// TIA Portal V20 export
// export: Created 2025-12-01T14:57:36.0041783Z, ExportSetting None, DisplayName Totally Integrated Automation Portal, DisplayVersion V20 Update 3, DisplayName TIA Portal Openness, DisplayVersion V20 Update 3, DisplayName TIA Portal Version Control Interface, DisplayVersion V20 Update 3, DisplayName STEP 7 Professional, DisplayVersion V20 Update 3, DisplayName STEP 7 Safety, DisplayVersion V20 Update 2, DisplayName WinCC Basic/Comfort/Advanced, DisplayVersion V20 Update 3, DisplayName WinCC Professional, DisplayVersion V20 Update 3, DisplayName WinCC Unified, DisplayVersion V20 Update 3
FUNCTION_BLOCK "FB984_Control_i950_ELEV / VTD"   // FB984, LAD
{ S7_Optimized_Access := 'FALSE' }
// stored: AutoNumber false, SetENOAutomatically false
   VAR_INPUT
      NumDispositivo : UInt;   // Numero de Maquina
      Error_Tx : Bool;
      Protusion : Bool;
      OrdenPosicion : Bool;
      "Avance-Subir" : Bool;
      "Retroceso-Bajar" : Bool;
      ConsignaPosicion : Real;
      SHome_Available : Bool;
      SHome_Activated : Bool;
   END_VAR
   VAR_OUTPUT
      PosicionActual : Real;
      VelocidadActual : Real;   // Velocidad Actual
      EnPosicion : Bool;   // Posicion OK de la Orden
      SHome_Start : Bool;   // Inicio Homing de la tarjeta SRM
      SHome_Load : Bool;   // Confirmacion de la tarjeta SRM
      Freno : Bool;
   END_VAR
   VAR
      TMP_Rearme { S7_SetPoint := 'True'} : TOF_TIME;
      TEspera_ET04Ref { S7_SetPoint := 'True'} : TON_TIME;
      TEspera_ET05Ref { S7_SetPoint := 'True'} : TON_TIME;
      TEspera_ET00 { S7_SetPoint := 'True'} : TON_TIME;
      PosicionOrden { S7_SetPoint := 'True'} : Real;
      ConsignaVelocidad : Real;
      ET_00 { S7_SetPoint := 'True'} : Bool;
      ET_01 : Bool;
      ET_02 : Bool;
      ET_03Ref : Bool;
      ET_04Ref : Bool;
      ET_05Ref : Bool;
      ET_06Ref : Bool;
      Rem_MesaDestino : UInt;
   END_VAR
   VAR_TEMP
      EstadoZona : "EstadoZona";   // Estado de la Zona
      EstadoMAQ : "EstadoMaquina_Variador_i950";
      NumMaquina : UInt;
      Byte0 : Int;
      Byte1 : Int;
      Byte2 : Int;
      Byte3 : Int;
      Direccion_Pos_Actual : DInt;
      Direccion_Velocity : DInt;
      Direccion_Position : DInt;
      DireccionCorriente : DInt;
      Acele : DInt;
      Dece : DInt;
      Jerk : DInt;
      Torque : DInt;
      DirInicial : Int;   // Dirección inicio periferia
      "ACC (m/s2)" : Real;
      "DCC(m/s2)" : Real;
      "VelocidadAuto(m/s)" : Real;
      "VelocidadHoming(m/s)" : Real;
      "PosicionHorming(mm)" : Real;
      VarReal : Real;
      Nodo : Int;   // Numero de Maquina
      VReal : DWord;
      VelocityAuto : DInt;
      VelocityHoming : DInt;
   END_VAR
   VAR_TEMP   // added for the SCL form of the ladder/FBD networks
      _w1 : Bool;
   END_VAR
BEGIN

REGION Network 1: Recoger Variables
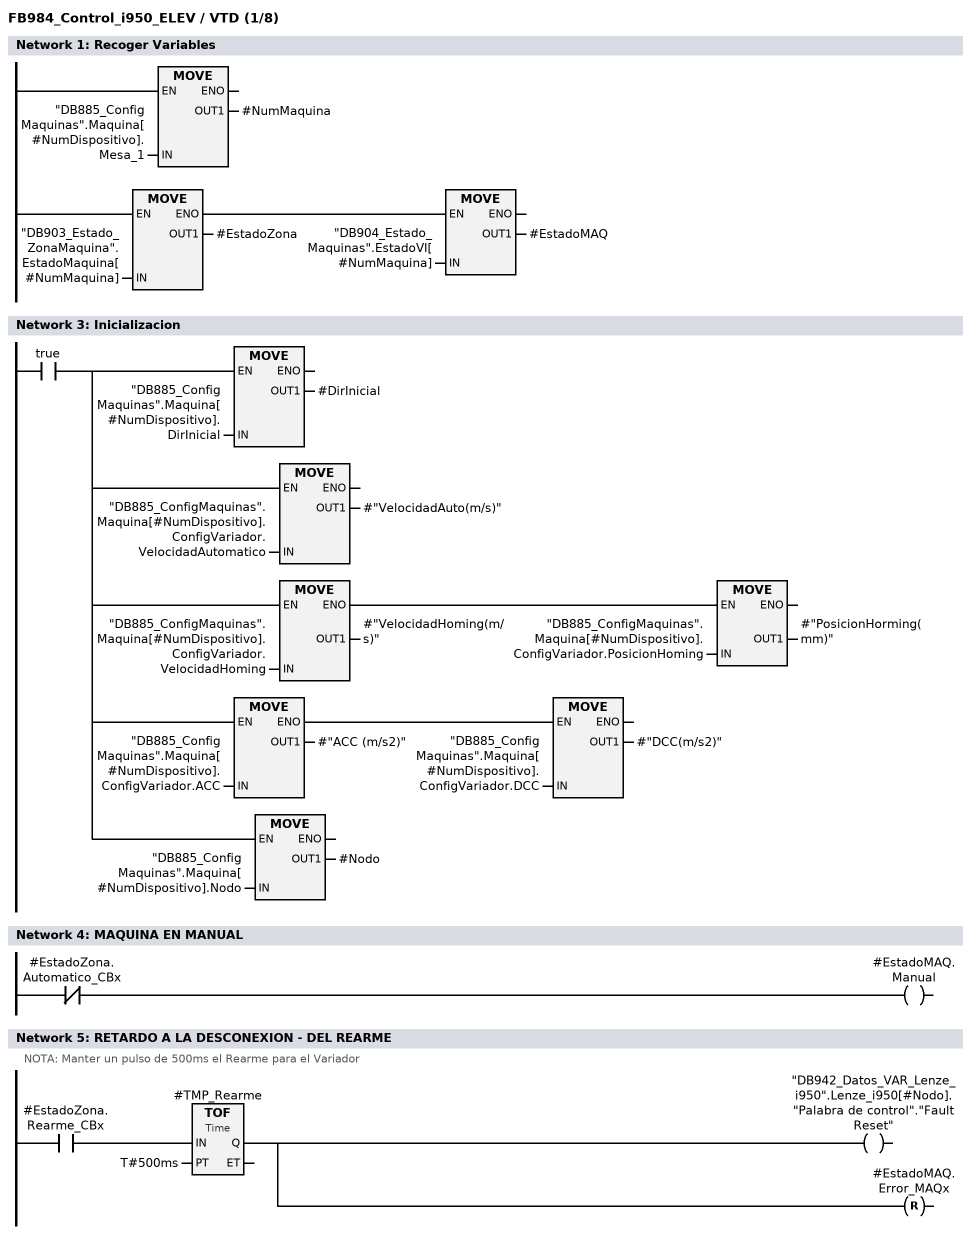
   RUNG wire#powerrail
      Move(in := "DB885_ConfigMaquinas".Maquina[#NumDispositivo].Mesa_1, out1 => #NumMaquina)
   END_RUNG
   RUNG wire#powerrail
      Move(in := "DB903_Estado_ZonaMaquina".EstadoMaquina[#NumMaquina], out1 => #EstadoZona)
      Move(in := "DB904_Estado_Maquinas".EstadoVI[#NumMaquina], out1 => #EstadoMAQ)
   END_RUNG
   // the same network as SCL:
   #NumMaquina := "DB885_ConfigMaquinas".Maquina[#NumDispositivo].Mesa_1;
   #EstadoZona := "DB903_Estado_ZonaMaquina".EstadoMaquina[#NumMaquina];
   #EstadoMAQ := "DB904_Estado_Maquinas".EstadoVI[#NumMaquina];
END_REGION

REGION Network 2: >>>>>>>>>>>>>>>>>>>>>>>>>>>>>>>>>>>>>>>>>>>>>>>>>>>>>>>>>>>>>>>>>>>>>>>
END_REGION

REGION Network 3: Inicializacion
   RUNG wire#powerrail
      Contact( true )
      wire#w1
      Move(in := "DB885_ConfigMaquinas".Maquina[#NumDispositivo].DirInicial, out1 => #DirInicial)
   END_RUNG
   RUNG wire#w1
      Move(in := "DB885_ConfigMaquinas".Maquina[#NumDispositivo].ConfigVariador.VelocidadAutomatico, out1 => #"VelocidadAuto(m/s)")
   END_RUNG
   RUNG wire#w1
      Move(in := "DB885_ConfigMaquinas".Maquina[#NumDispositivo].ConfigVariador.VelocidadHoming, out1 => #"VelocidadHoming(m/s)")
      Move(in := "DB885_ConfigMaquinas".Maquina[#NumDispositivo].ConfigVariador.PosicionHoming, out1 => #"PosicionHorming(mm)")
   END_RUNG
   RUNG wire#w1
      Move(in := "DB885_ConfigMaquinas".Maquina[#NumDispositivo].ConfigVariador.ACC, out1 => #"ACC (m/s2)")
      Move(in := "DB885_ConfigMaquinas".Maquina[#NumDispositivo].ConfigVariador.DCC, out1 => #"DCC(m/s2)")
   END_RUNG
   RUNG wire#w1
      Move(in := "DB885_ConfigMaquinas".Maquina[#NumDispositivo].Nodo, out1 => #Nodo)
   END_RUNG
   // the same network as SCL:
   IF true THEN
       #DirInicial := "DB885_ConfigMaquinas".Maquina[#NumDispositivo].DirInicial;
       #"VelocidadAuto(m/s)" := "DB885_ConfigMaquinas".Maquina[#NumDispositivo].ConfigVariador.VelocidadAutomatico;
       #"VelocidadHoming(m/s)" := "DB885_ConfigMaquinas".Maquina[#NumDispositivo].ConfigVariador.VelocidadHoming;
       #"PosicionHorming(mm)" := "DB885_ConfigMaquinas".Maquina[#NumDispositivo].ConfigVariador.PosicionHoming;
       #"ACC (m/s2)" := "DB885_ConfigMaquinas".Maquina[#NumDispositivo].ConfigVariador.ACC;
       #"DCC(m/s2)" := "DB885_ConfigMaquinas".Maquina[#NumDispositivo].ConfigVariador.DCC;
       #Nodo := "DB885_ConfigMaquinas".Maquina[#NumDispositivo].Nodo;
   END_IF;
END_REGION

REGION Network 4: MAQUINA EN MANUAL
   RUNG wire#powerrail
      I_Contact( #EstadoZona.Automatico_CBx )
      Coil( #EstadoMAQ.Manual )
   END_RUNG
   // the same network as SCL:
   #EstadoMAQ.Manual := NOT #EstadoZona.Automatico_CBx;
END_REGION

REGION Network 5: RETARDO A LA DESCONEXION - DEL REARME
   // NOTA: Manter un pulso de 500ms el Rearme para el Variador
   RUNG wire#powerrail
      Contact( #EstadoZona.Rearme_CBx )
      { S7_Templates := "time_type := Time" } #TMP_Rearme.TOF(pt := T#500ms, et =>)
      wire#w1
      Coil( "DB942_Datos_VAR_Lenze_i950".Lenze_i950[#Nodo]."Palabra de control"."Fault Reset" )
   END_RUNG
   RUNG wire#w1
      R_Coil( #EstadoMAQ.Error_MAQx )
   END_RUNG
   // the same network as SCL:
   #TMP_Rearme(IN := #EstadoZona.Rearme_CBx, PT := T#500ms);   // TOF
   "DB942_Datos_VAR_Lenze_i950".Lenze_i950[#Nodo]."Palabra de control"."Fault Reset" := #TMP_Rearme.Q;
   IF #TMP_Rearme.Q THEN #EstadoMAQ.Error_MAQx := FALSE; END_IF;
END_REGION

REGION Network 6 (SCL): Direcciones
   #Byte0 := #DirInicial;
   #Byte1 := #DirInicial + 1;
   #Byte2 := #DirInicial + 2;
   #Byte3 := #DirInicial + 3;
   #Direccion_Pos_Actual := #DirInicial + 12;
   #Direccion_Velocity := #DirInicial + 8;
   #Direccion_Position := #DirInicial + 12;
   #DireccionCorriente := #DirInicial + 24;
   #Acele := #DirInicial + 16;
   #Dece := #DirInicial + 20;
   #Jerk := #DirInicial + 24;
   #Torque := #DirInicial + 28;
END_REGION

REGION Network 7 (SCL): Lectura de variables del Variador
   //Leo las variables que nos interesan

   "DB942_Datos_VAR_Lenze_i950".Lenze_i950[#Nodo]."Estatus variador"."Positioning Profile Done" := PEEK_BOOL(area := 16#81, dbNumber := 0, byteOffset := #Byte1, bitOffset := 5);
   "DB942_Datos_VAR_Lenze_i950".Lenze_i950[#Nodo]."Estatus variador"."Target Reached" := PEEK_BOOL(area := 16#81, dbNumber := 0, byteOffset := #Byte2, bitOffset := 2);
   "DB942_Datos_VAR_Lenze_i950".Lenze_i950[#Nodo]."Estatus variador"."STO Active" := PEEK_BOOL(area := 16#81, dbNumber := 0, byteOffset := #Byte2, bitOffset := 7);
   "DB942_Datos_VAR_Lenze_i950".Lenze_i950[#Nodo]."Estatus variador"."Operation Enabled" := PEEK_BOOL(area := 16#81, dbNumber := 0, byteOffset := #Byte3, bitOffset := 2);
   "DB942_Datos_VAR_Lenze_i950".Lenze_i950[#Nodo]."Estatus variador"."Drive Fault" := PEEK_BOOL(area := 16#81, dbNumber := 0, byteOffset := #Byte3, bitOffset := 3);
   "DB942_Datos_VAR_Lenze_i950".Lenze_i950[#Nodo]."Estatus variador"."Drive Homed" := PEEK_BOOL(area := 16#81, dbNumber := 0, byteOffset := #Byte3, bitOffset := 4);
   "DB942_Datos_VAR_Lenze_i950".Lenze_i950[#Nodo]."Estatus variador"."Jogging Busy" := PEEK_BOOL(area := 16#81, dbNumber := 0, byteOffset := #Byte3, bitOffset := 6);
   "DB942_Datos_VAR_Lenze_i950".Lenze_i950[#Nodo].Velocity := PEEK_DWORD(area := 16#81, dbNumber := 0, byteOffset := #Direccion_Velocity);
   "DB942_Datos_VAR_Lenze_i950".Lenze_i950[#Nodo].Actual_Position := PEEK_DWORD(area := 16#81, dbNumber := 0, byteOffset := #Direccion_Pos_Actual);
   "DB942_Datos_VAR_Lenze_i950".Lenze_i950[#Nodo]."Corriente%" := PEEK_DWORD(area := 16#81, dbNumber := 0, byteOffset := #DireccionCorriente);
END_REGION

REGION Network 8: Captura de la corriente
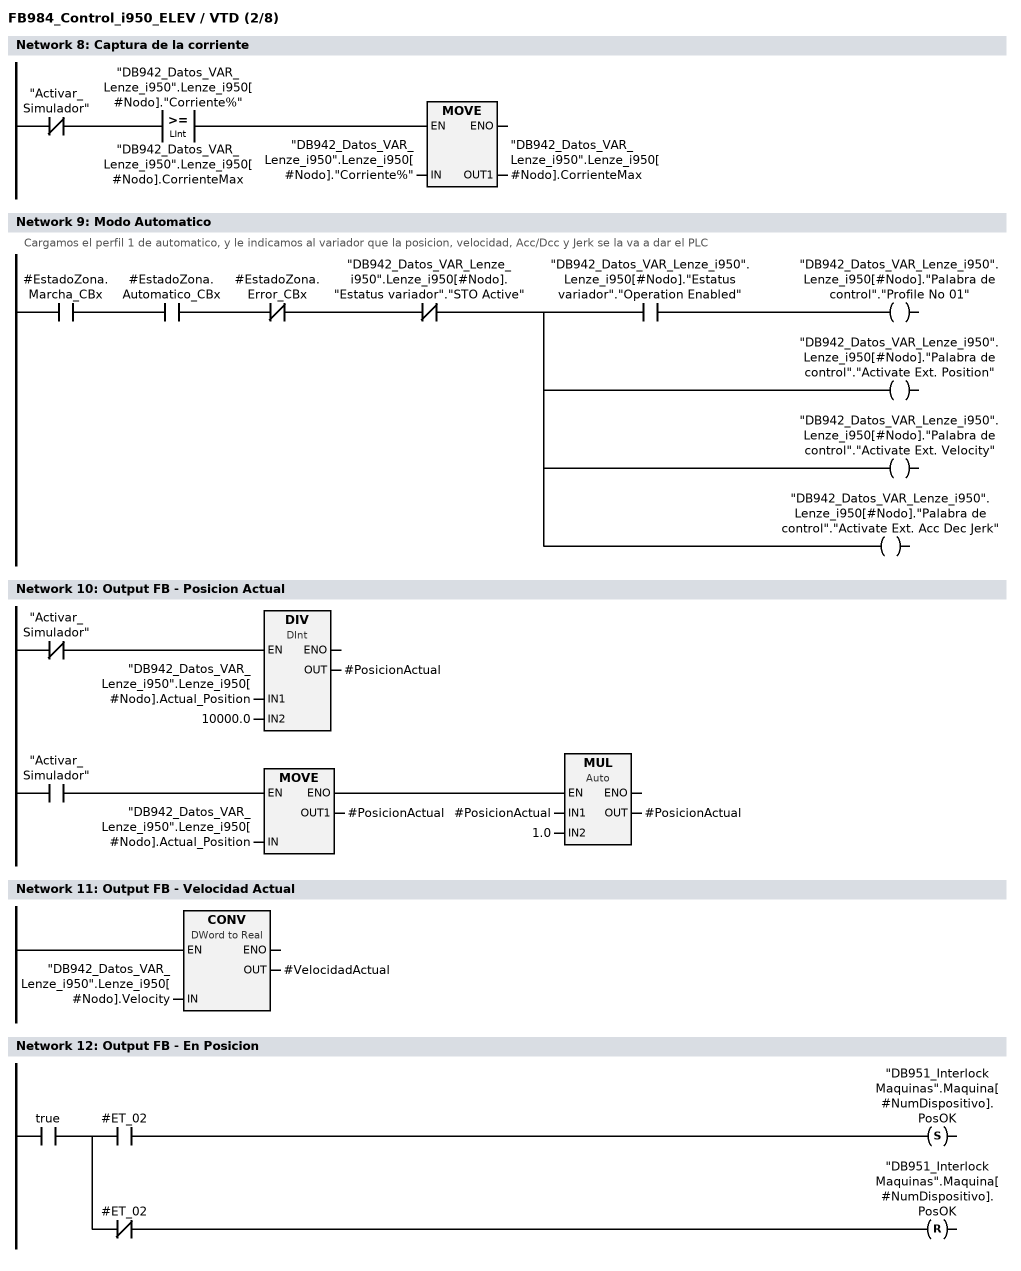
   RUNG wire#powerrail
      I_Contact( "Activar_Simulador" )
      { S7_Templates := "SrcType := LInt" } GE_Contact(in1 := "DB942_Datos_VAR_Lenze_i950".Lenze_i950[#Nodo]."Corriente%", in2 := "DB942_Datos_VAR_Lenze_i950".Lenze_i950[#Nodo].CorrienteMax)
      Move(in := "DB942_Datos_VAR_Lenze_i950".Lenze_i950[#Nodo]."Corriente%", out1 => "DB942_Datos_VAR_Lenze_i950".Lenze_i950[#Nodo].CorrienteMax)
   END_RUNG
   // the same network as SCL:
   IF NOT "Activar_Simulador" AND ("DB942_Datos_VAR_Lenze_i950".Lenze_i950[#Nodo]."Corriente%" >= "DB942_Datos_VAR_Lenze_i950".Lenze_i950[#Nodo].CorrienteMax) THEN
       "DB942_Datos_VAR_Lenze_i950".Lenze_i950[#Nodo].CorrienteMax := "DB942_Datos_VAR_Lenze_i950".Lenze_i950[#Nodo]."Corriente%";
   END_IF;
END_REGION

REGION Network 9: Modo Automatico
   // Cargamos el perfil 1 de automatico, y le indicamos al variador que la posicion, velocidad, Acc/Dcc y Jerk se la va a dar el PLC
   RUNG wire#powerrail
      Contact( #EstadoZona.Marcha_CBx )
      Contact( #EstadoZona.Automatico_CBx )
      I_Contact( #EstadoZona.Error_CBx )
      I_Contact( "DB942_Datos_VAR_Lenze_i950".Lenze_i950[#Nodo]."Estatus variador"."STO Active" )
      wire#w1
      Contact( "DB942_Datos_VAR_Lenze_i950".Lenze_i950[#Nodo]."Estatus variador"."Operation Enabled" )
      Coil( "DB942_Datos_VAR_Lenze_i950".Lenze_i950[#Nodo]."Palabra de control"."Profile No 01" )
   END_RUNG
   RUNG wire#w1
      Coil( "DB942_Datos_VAR_Lenze_i950".Lenze_i950[#Nodo]."Palabra de control"."Activate Ext. Position" )
   END_RUNG
   RUNG wire#w1
      Coil( "DB942_Datos_VAR_Lenze_i950".Lenze_i950[#Nodo]."Palabra de control"."Activate Ext. Velocity" )
   END_RUNG
   RUNG wire#w1
      Coil( "DB942_Datos_VAR_Lenze_i950".Lenze_i950[#Nodo]."Palabra de control"."Activate Ext. Acc Dec Jerk" )
   END_RUNG
   // the same network as SCL:
   #_w1 := #EstadoZona.Marcha_CBx AND #EstadoZona.Automatico_CBx AND NOT #EstadoZona.Error_CBx AND NOT "DB942_Datos_VAR_Lenze_i950".Lenze_i950[#Nodo]."Estatus variador"."STO Active";
   "DB942_Datos_VAR_Lenze_i950".Lenze_i950[#Nodo]."Palabra de control"."Profile No 01" := #_w1 AND "DB942_Datos_VAR_Lenze_i950".Lenze_i950[#Nodo]."Estatus variador"."Operation Enabled";
   "DB942_Datos_VAR_Lenze_i950".Lenze_i950[#Nodo]."Palabra de control"."Activate Ext. Position" := #_w1;
   "DB942_Datos_VAR_Lenze_i950".Lenze_i950[#Nodo]."Palabra de control"."Activate Ext. Velocity" := #_w1;
   "DB942_Datos_VAR_Lenze_i950".Lenze_i950[#Nodo]."Palabra de control"."Activate Ext. Acc Dec Jerk" := #_w1;
END_REGION

REGION Network 10: Output FB - Posicion Actual
   RUNG wire#powerrail
      I_Contact( "Activar_Simulador" )
      { S7_Templates := "SrcType := DInt" } Div(in1 := "DB942_Datos_VAR_Lenze_i950".Lenze_i950[#Nodo].Actual_Position, in2 := 10000.0, out => #PosicionActual)
   END_RUNG
   RUNG wire#powerrail
      Contact( "Activar_Simulador" )
      Move(in := "DB942_Datos_VAR_Lenze_i950".Lenze_i950[#Nodo].Actual_Position, out1 => #PosicionActual)
      Mul(in1 := #PosicionActual, in2 := 1.0, out => #PosicionActual)
   END_RUNG
   // the same network as SCL:
   IF NOT "Activar_Simulador" THEN
       #PosicionActual := "DB942_Datos_VAR_Lenze_i950".Lenze_i950[#Nodo].Actual_Position / 10000.0;
   END_IF;
   IF "Activar_Simulador" THEN
       #PosicionActual := "DB942_Datos_VAR_Lenze_i950".Lenze_i950[#Nodo].Actual_Position;
       #PosicionActual := #PosicionActual * 1.0;
   END_IF;
END_REGION

REGION Network 11: Output FB - Velocidad Actual
   RUNG wire#powerrail
      { S7_Templates := "[SrcType := DWord, DestType := Real]" } Convert(in := "DB942_Datos_VAR_Lenze_i950".Lenze_i950[#Nodo].Velocity, out => #VelocidadActual)
   END_RUNG
   // the same network as SCL:
   #VelocidadActual := DWORD_TO_REAL("DB942_Datos_VAR_Lenze_i950".Lenze_i950[#Nodo].Velocity);
END_REGION

REGION Network 12: Output FB - En Posicion
   RUNG wire#powerrail
      Contact( true )
      wire#w1
      Contact( #ET_02 )
      S_Coil( "DB951_InterlockMaquinas".Maquina[#NumDispositivo].PosOK )
   END_RUNG
   RUNG wire#w1
      I_Contact( #ET_02 )
      R_Coil( "DB951_InterlockMaquinas".Maquina[#NumDispositivo].PosOK )
   END_RUNG
   // the same network as SCL:
   IF true AND #ET_02 THEN "DB951_InterlockMaquinas".Maquina[#NumDispositivo].PosOK := TRUE; END_IF;
   IF true AND NOT #ET_02 THEN "DB951_InterlockMaquinas".Maquina[#NumDispositivo].PosOK := FALSE; END_IF;
END_REGION

REGION Network 13: Consigna de Velocidad
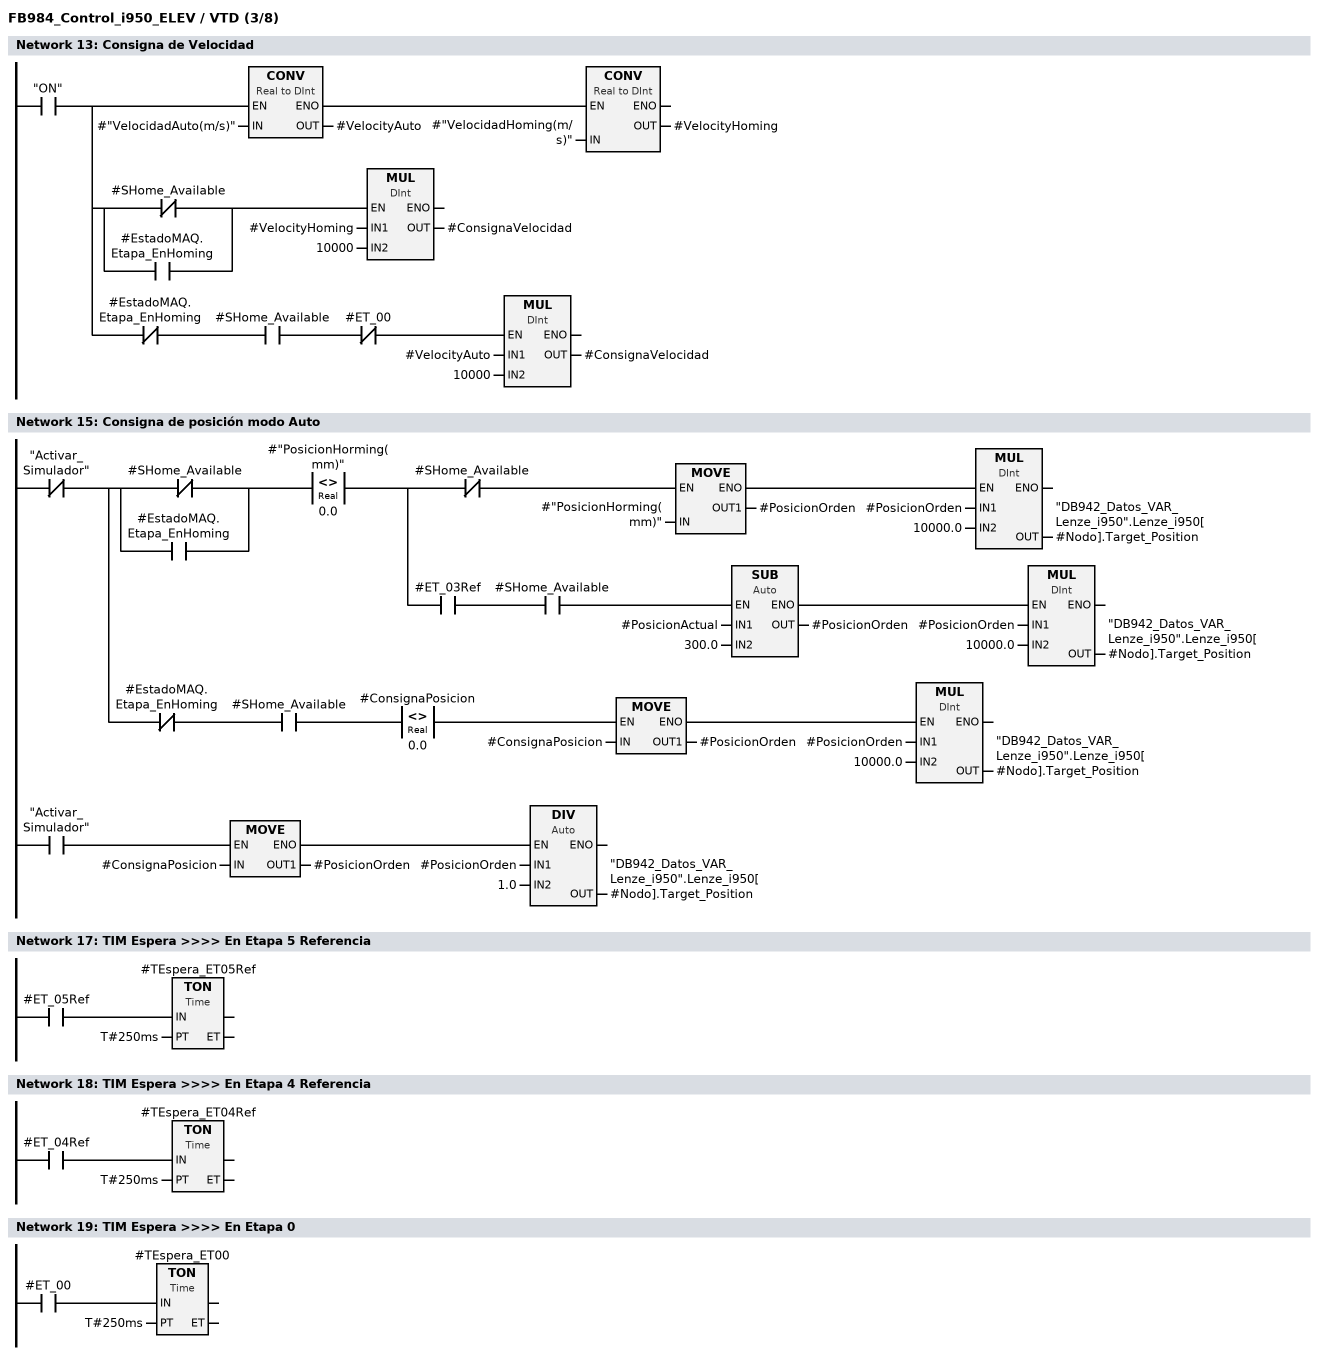
   RUNG wire#powerrail
      Contact( "ON" )
      wire#w1
      { S7_Templates := "[SrcType := Real, DestType := DInt]" } Convert(in := #"VelocidadAuto(m/s)", out => #VelocityAuto)
      { S7_Templates := "[SrcType := Real, DestType := DInt]" } Convert(in := #"VelocidadHoming(m/s)", out => #VelocityHoming)
   END_RUNG
   RUNG wire#w1
      I_Contact( #SHome_Available )
      wire#w2
      { S7_Templates := "SrcType := DInt" } Mul(in1 := #VelocityHoming, in2 := 10000, out => #ConsignaVelocidad)
   END_RUNG
   RUNG wire#w1
      Contact( #EstadoMAQ.Etapa_EnHoming )
   END_RUNG wire#w2
   RUNG wire#w1
      I_Contact( #EstadoMAQ.Etapa_EnHoming )
      Contact( #SHome_Available )
      I_Contact( #ET_00 )
      { S7_Templates := "SrcType := DInt" } Mul(in1 := #VelocityAuto, in2 := 10000, out => #ConsignaVelocidad)
   END_RUNG
   // the same network as SCL:
   IF "ON" THEN
       #VelocityAuto := REAL_TO_DINT(#"VelocidadAuto(m/s)");
       #VelocityHoming := REAL_TO_DINT(#"VelocidadHoming(m/s)");
   END_IF;
   IF "ON" AND (NOT #SHome_Available OR #EstadoMAQ.Etapa_EnHoming) THEN
       #ConsignaVelocidad := #VelocityHoming * 10000;
   END_IF;
   IF "ON" AND NOT #EstadoMAQ.Etapa_EnHoming AND #SHome_Available AND NOT #ET_00 THEN
       #ConsignaVelocidad := #VelocityAuto * 10000;
   END_IF;
END_REGION

REGION Network 14 (SCL): Aceleración y Deceleración
   "DB942_Datos_VAR_Lenze_i950".Lenze_i950[#Nodo].ACC := REAL_TO_DINT (#"ACC (m/s2)" * 100);
   "DB942_Datos_VAR_Lenze_i950".Lenze_i950[#Nodo].DCC  := REAL_TO_DINT(#"DCC(m/s2)" * 100);
END_REGION

REGION Network 15: Consigna de posición modo Auto
   RUNG wire#powerrail
      I_Contact( "Activar_Simulador" )
      wire#w1
      I_Contact( #SHome_Available )
      wire#w2
      { S7_Templates := "SrcType := Real" } NE_Contact(in1 := #"PosicionHorming(mm)", in2 := 0.0)
      wire#w3
      I_Contact( #SHome_Available )
      Move(in := #"PosicionHorming(mm)", out1 => #PosicionOrden)
      { S7_Templates := "SrcType := DInt" } Mul(in1 := #PosicionOrden, in2 := 10000.0, out => "DB942_Datos_VAR_Lenze_i950".Lenze_i950[#Nodo].Target_Position)
   END_RUNG
   RUNG wire#w1
      Contact( #EstadoMAQ.Etapa_EnHoming )
   END_RUNG wire#w2
   RUNG wire#w3
      Contact( #ET_03Ref )
      Contact( #SHome_Available )
      Sub(in1 := #PosicionActual, in2 := 300.0, out => #PosicionOrden)
      { S7_Templates := "SrcType := DInt" } Mul(in1 := #PosicionOrden, in2 := 10000.0, out => "DB942_Datos_VAR_Lenze_i950".Lenze_i950[#Nodo].Target_Position)
   END_RUNG
   RUNG wire#w1
      I_Contact( #EstadoMAQ.Etapa_EnHoming )
      Contact( #SHome_Available )
      { S7_Templates := "SrcType := Real" } NE_Contact(in1 := #ConsignaPosicion, in2 := 0.0)
      Move(in := #ConsignaPosicion, out1 => #PosicionOrden)
      { S7_Templates := "SrcType := DInt" } Mul(in1 := #PosicionOrden, in2 := 10000.0, out => "DB942_Datos_VAR_Lenze_i950".Lenze_i950[#Nodo].Target_Position)
   END_RUNG
   RUNG wire#powerrail
      Contact( "Activar_Simulador" )
      Move(in := #ConsignaPosicion, out1 => #PosicionOrden)
      Div(in1 := #PosicionOrden, in2 := 1.0, out => "DB942_Datos_VAR_Lenze_i950".Lenze_i950[#Nodo].Target_Position)
   END_RUNG
   // the same network as SCL:
   #_w1 := NOT "Activar_Simulador" AND (NOT #SHome_Available OR #EstadoMAQ.Etapa_EnHoming) AND (#"PosicionHorming(mm)" <> 0.0);
   IF #_w1 AND NOT #SHome_Available THEN
       #PosicionOrden := #"PosicionHorming(mm)";
       "DB942_Datos_VAR_Lenze_i950".Lenze_i950[#Nodo].Target_Position := #PosicionOrden * 10000.0;
   END_IF;
   IF #_w1 AND #ET_03Ref AND #SHome_Available THEN
       #PosicionOrden := #PosicionActual - 300.0;
       "DB942_Datos_VAR_Lenze_i950".Lenze_i950[#Nodo].Target_Position := #PosicionOrden * 10000.0;
   END_IF;
   IF NOT "Activar_Simulador" AND NOT #EstadoMAQ.Etapa_EnHoming AND #SHome_Available AND (#ConsignaPosicion <> 0.0) THEN
       #PosicionOrden := #ConsignaPosicion;
       "DB942_Datos_VAR_Lenze_i950".Lenze_i950[#Nodo].Target_Position := #PosicionOrden * 10000.0;
   END_IF;
   IF "Activar_Simulador" THEN
       #PosicionOrden := #ConsignaPosicion;
       "DB942_Datos_VAR_Lenze_i950".Lenze_i950[#Nodo].Target_Position := #PosicionOrden / 1.0;
   END_IF;
END_REGION

REGION Network 16: >>>>>>>>>>>>>>>>>>>>>>>>>>>>>>>>>>>>>>>>>>>>>>>>>>>>>>>>>>>>>>>>>>>>>>>>>>>>>
END_REGION

REGION Network 17: TIM Espera >>>> En Etapa 5 Referencia
   RUNG wire#powerrail
      Contact( #ET_05Ref )
      { S7_Templates := "time_type := Time" } #TEspera_ET05Ref.TON(pt := T#250ms, et =>)
   END_RUNG
   // the same network as SCL:
   #TEspera_ET05Ref(IN := #ET_05Ref, PT := T#250ms);   // TON
END_REGION

REGION Network 18: TIM Espera >>>> En Etapa 4 Referencia
   RUNG wire#powerrail
      Contact( #ET_04Ref )
      { S7_Templates := "time_type := Time" } #TEspera_ET04Ref.TON(pt := T#250ms, et =>)
   END_RUNG
   // the same network as SCL:
   #TEspera_ET04Ref(IN := #ET_04Ref, PT := T#250ms);   // TON
END_REGION

REGION Network 19: TIM Espera >>>> En Etapa 0
   RUNG wire#powerrail
      Contact( #ET_00 )
      { S7_Templates := "time_type := Time" } #TEspera_ET00.TON(pt := T#250ms, et =>)
   END_RUNG
   // the same network as SCL:
   #TEspera_ET00(IN := #ET_00, PT := T#250ms);   // TON
END_REGION

REGION Network 20: >>>>>>>>>>>>>>>>>>>>>>>>>>>>>>>>>>>>>>>>>>>>>>>>>>>>>>>>>>>>>>>>>>>>>>>>>>>>>
END_REGION

REGION Network 21: ET06Ref - Fin Homing
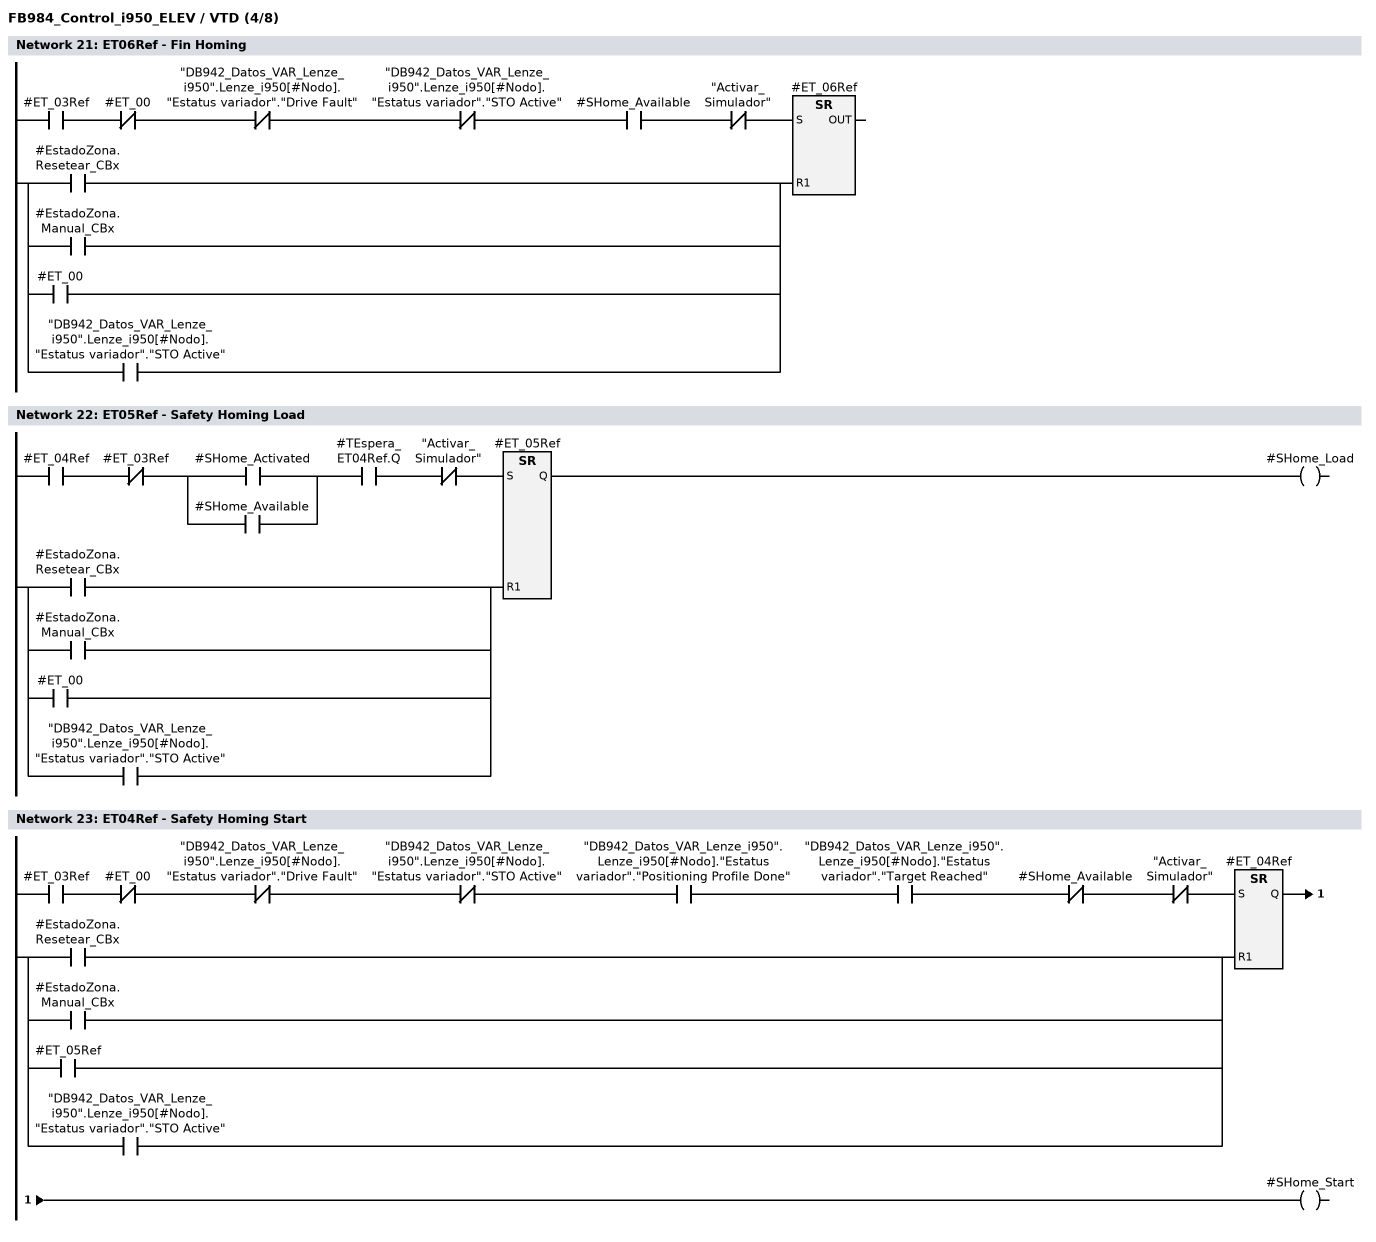
   RUNG wire#powerrail
      Contact( #ET_03Ref )
      I_Contact( #ET_00 )
      I_Contact( "DB942_Datos_VAR_Lenze_i950".Lenze_i950[#Nodo]."Estatus variador"."Drive Fault" )
      I_Contact( "DB942_Datos_VAR_Lenze_i950".Lenze_i950[#Nodo]."Estatus variador"."STO Active" )
      Contact( #SHome_Available )
      I_Contact( "Activar_Simulador" )
      S_SR(operand := #ET_06Ref, r1 := wire#w1)
   END_RUNG
   RUNG wire#powerrail
      Contact( #EstadoZona.Resetear_CBx )
   END_RUNG wire#w1
   RUNG wire#powerrail
      Contact( #EstadoZona.Manual_CBx )
   END_RUNG wire#w1
   RUNG wire#powerrail
      Contact( #ET_00 )
   END_RUNG wire#w1
   RUNG wire#powerrail
      Contact( "DB942_Datos_VAR_Lenze_i950".Lenze_i950[#Nodo]."Estatus variador"."STO Active" )
   END_RUNG wire#w1
   // the same network as SCL:
   IF #ET_03Ref AND NOT #ET_00 AND NOT "DB942_Datos_VAR_Lenze_i950".Lenze_i950[#Nodo]."Estatus variador"."Drive Fault" AND NOT "DB942_Datos_VAR_Lenze_i950".Lenze_i950[#Nodo]."Estatus variador"."STO Active" AND #SHome_Available AND NOT "Activar_Simulador" THEN
       #ET_06Ref := TRUE;   // SR flip-flop
   END_IF;
   IF #EstadoZona.Resetear_CBx OR #EstadoZona.Manual_CBx OR #ET_00 OR "DB942_Datos_VAR_Lenze_i950".Lenze_i950[#Nodo]."Estatus variador"."STO Active" THEN
       #ET_06Ref := FALSE;
   END_IF;
END_REGION

REGION Network 22: ET05Ref - Safety Homing Load
   RUNG wire#powerrail
      Contact( #ET_04Ref )
      I_Contact( #ET_03Ref )
      wire#w1
      Contact( #SHome_Activated )
      wire#w2
      Contact( #TEspera_ET04Ref.Q )
      I_Contact( "Activar_Simulador" )
      S_SR(operand := #ET_05Ref, r1 := wire#w3)
      Coil( #SHome_Load )
   END_RUNG
   RUNG wire#w1
      Contact( #SHome_Available )
   END_RUNG wire#w2
   RUNG wire#powerrail
      Contact( #EstadoZona.Resetear_CBx )
   END_RUNG wire#w3
   RUNG wire#powerrail
      Contact( #EstadoZona.Manual_CBx )
   END_RUNG wire#w3
   RUNG wire#powerrail
      Contact( #ET_00 )
   END_RUNG wire#w3
   RUNG wire#powerrail
      Contact( "DB942_Datos_VAR_Lenze_i950".Lenze_i950[#Nodo]."Estatus variador"."STO Active" )
   END_RUNG wire#w3
   // the same network as SCL:
   IF #ET_04Ref AND NOT #ET_03Ref AND (#SHome_Activated OR #SHome_Available) AND #TEspera_ET04Ref.Q AND NOT "Activar_Simulador" THEN
       #ET_05Ref := TRUE;   // SR flip-flop
   END_IF;
   IF #EstadoZona.Resetear_CBx OR #EstadoZona.Manual_CBx OR #ET_00 OR "DB942_Datos_VAR_Lenze_i950".Lenze_i950[#Nodo]."Estatus variador"."STO Active" THEN
       #ET_05Ref := FALSE;
   END_IF;
   #SHome_Load := #ET_05Ref;
END_REGION

REGION Network 23: ET04Ref - Safety Homing Start
   RUNG wire#powerrail
      Contact( #ET_03Ref )
      I_Contact( #ET_00 )
      I_Contact( "DB942_Datos_VAR_Lenze_i950".Lenze_i950[#Nodo]."Estatus variador"."Drive Fault" )
      I_Contact( "DB942_Datos_VAR_Lenze_i950".Lenze_i950[#Nodo]."Estatus variador"."STO Active" )
      Contact( "DB942_Datos_VAR_Lenze_i950".Lenze_i950[#Nodo]."Estatus variador"."Positioning Profile Done" )
      Contact( "DB942_Datos_VAR_Lenze_i950".Lenze_i950[#Nodo]."Estatus variador"."Target Reached" )
      I_Contact( #SHome_Available )
      I_Contact( "Activar_Simulador" )
      S_SR(operand := #ET_04Ref, r1 := wire#w1)
      Coil( #SHome_Start )
   END_RUNG
   RUNG wire#powerrail
      Contact( #EstadoZona.Resetear_CBx )
   END_RUNG wire#w1
   RUNG wire#powerrail
      Contact( #EstadoZona.Manual_CBx )
   END_RUNG wire#w1
   RUNG wire#powerrail
      Contact( #ET_05Ref )
   END_RUNG wire#w1
   RUNG wire#powerrail
      Contact( "DB942_Datos_VAR_Lenze_i950".Lenze_i950[#Nodo]."Estatus variador"."STO Active" )
   END_RUNG wire#w1
   // the same network as SCL:
   IF #ET_03Ref AND NOT #ET_00 AND NOT "DB942_Datos_VAR_Lenze_i950".Lenze_i950[#Nodo]."Estatus variador"."Drive Fault" AND NOT "DB942_Datos_VAR_Lenze_i950".Lenze_i950[#Nodo]."Estatus variador"."STO Active" AND "DB942_Datos_VAR_Lenze_i950".Lenze_i950[#Nodo]."Estatus variador"."Positioning Profile Done" AND "DB942_Datos_VAR_Lenze_i950".Lenze_i950[#Nodo]."Estatus variador"."Target Reached" AND NOT #SHome_Available AND NOT "Activar_Simulador" THEN
       #ET_04Ref := TRUE;   // SR flip-flop
   END_IF;
   IF #EstadoZona.Resetear_CBx OR #EstadoZona.Manual_CBx OR #ET_05Ref OR "DB942_Datos_VAR_Lenze_i950".Lenze_i950[#Nodo]."Estatus variador"."STO Active" THEN
       #ET_04Ref := FALSE;
   END_IF;
   #SHome_Start := #ET_04Ref;
END_REGION

REGION Network 24: ET03Ref - Safety Homing Posicionar
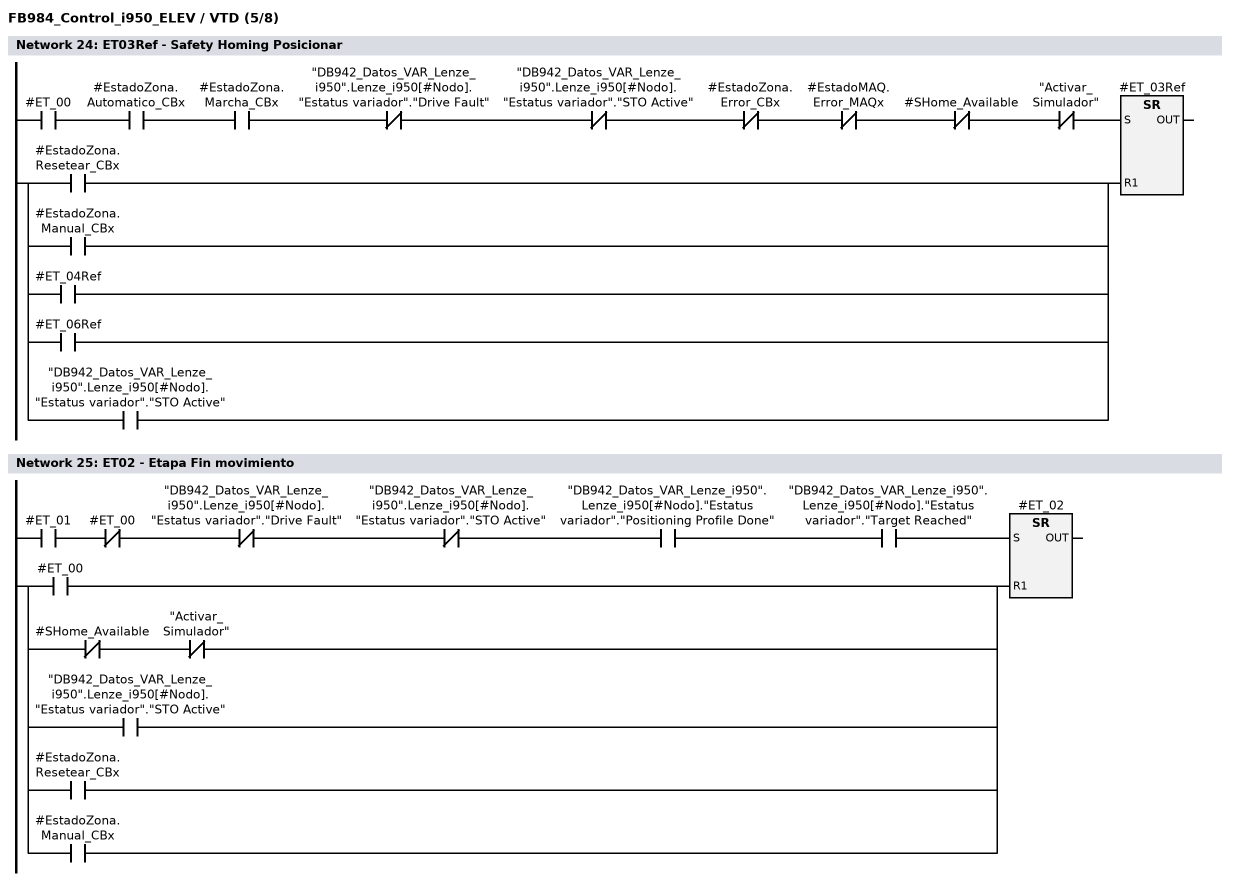
   RUNG wire#powerrail
      Contact( #ET_00 )
      Contact( #EstadoZona.Automatico_CBx )
      Contact( #EstadoZona.Marcha_CBx )
      I_Contact( "DB942_Datos_VAR_Lenze_i950".Lenze_i950[#Nodo]."Estatus variador"."Drive Fault" )
      I_Contact( "DB942_Datos_VAR_Lenze_i950".Lenze_i950[#Nodo]."Estatus variador"."STO Active" )
      I_Contact( #EstadoZona.Error_CBx )
      I_Contact( #EstadoMAQ.Error_MAQx )
      I_Contact( #SHome_Available )
      I_Contact( "Activar_Simulador" )
      S_SR(operand := #ET_03Ref, r1 := wire#w1)
   END_RUNG
   RUNG wire#powerrail
      Contact( #EstadoZona.Resetear_CBx )
   END_RUNG wire#w1
   RUNG wire#powerrail
      Contact( #EstadoZona.Manual_CBx )
   END_RUNG wire#w1
   RUNG wire#powerrail
      Contact( #ET_04Ref )
   END_RUNG wire#w1
   RUNG wire#powerrail
      Contact( #ET_06Ref )
   END_RUNG wire#w1
   RUNG wire#powerrail
      Contact( "DB942_Datos_VAR_Lenze_i950".Lenze_i950[#Nodo]."Estatus variador"."STO Active" )
   END_RUNG wire#w1
   // the same network as SCL:
   IF #ET_00 AND #EstadoZona.Automatico_CBx AND #EstadoZona.Marcha_CBx AND NOT "DB942_Datos_VAR_Lenze_i950".Lenze_i950[#Nodo]."Estatus variador"."Drive Fault" AND NOT "DB942_Datos_VAR_Lenze_i950".Lenze_i950[#Nodo]."Estatus variador"."STO Active" AND NOT #EstadoZona.Error_CBx AND NOT #EstadoMAQ.Error_MAQx AND NOT #SHome_Available AND NOT "Activar_Simulador" THEN
       #ET_03Ref := TRUE;   // SR flip-flop
   END_IF;
   IF #EstadoZona.Resetear_CBx OR #EstadoZona.Manual_CBx OR #ET_04Ref OR #ET_06Ref OR "DB942_Datos_VAR_Lenze_i950".Lenze_i950[#Nodo]."Estatus variador"."STO Active" THEN
       #ET_03Ref := FALSE;
   END_IF;
END_REGION

REGION Network 25: ET02 - Etapa Fin movimiento
   RUNG wire#powerrail
      Contact( #ET_01 )
      I_Contact( #ET_00 )
      I_Contact( "DB942_Datos_VAR_Lenze_i950".Lenze_i950[#Nodo]."Estatus variador"."Drive Fault" )
      I_Contact( "DB942_Datos_VAR_Lenze_i950".Lenze_i950[#Nodo]."Estatus variador"."STO Active" )
      Contact( "DB942_Datos_VAR_Lenze_i950".Lenze_i950[#Nodo]."Estatus variador"."Positioning Profile Done" )
      Contact( "DB942_Datos_VAR_Lenze_i950".Lenze_i950[#Nodo]."Estatus variador"."Target Reached" )
      S_SR(operand := #ET_02, r1 := wire#w1)
   END_RUNG
   RUNG wire#powerrail
      Contact( #ET_00 )
   END_RUNG wire#w1
   RUNG wire#powerrail
      I_Contact( #SHome_Available )
      I_Contact( "Activar_Simulador" )
   END_RUNG wire#w1
   RUNG wire#powerrail
      Contact( "DB942_Datos_VAR_Lenze_i950".Lenze_i950[#Nodo]."Estatus variador"."STO Active" )
   END_RUNG wire#w1
   RUNG wire#powerrail
      Contact( #EstadoZona.Resetear_CBx )
   END_RUNG wire#w1
   RUNG wire#powerrail
      Contact( #EstadoZona.Manual_CBx )
   END_RUNG wire#w1
   // the same network as SCL:
   IF #ET_01 AND NOT #ET_00 AND NOT "DB942_Datos_VAR_Lenze_i950".Lenze_i950[#Nodo]."Estatus variador"."Drive Fault" AND NOT "DB942_Datos_VAR_Lenze_i950".Lenze_i950[#Nodo]."Estatus variador"."STO Active" AND "DB942_Datos_VAR_Lenze_i950".Lenze_i950[#Nodo]."Estatus variador"."Positioning Profile Done" AND "DB942_Datos_VAR_Lenze_i950".Lenze_i950[#Nodo]."Estatus variador"."Target Reached" THEN
       #ET_02 := TRUE;   // SR flip-flop
   END_IF;
   IF #ET_00 OR (NOT #SHome_Available AND NOT "Activar_Simulador") OR "DB942_Datos_VAR_Lenze_i950".Lenze_i950[#Nodo]."Estatus variador"."STO Active" OR #EstadoZona.Resetear_CBx OR #EstadoZona.Manual_CBx THEN
       #ET_02 := FALSE;
   END_IF;
END_REGION

REGION Network 26: ET01 - Etapa movimiento en curso
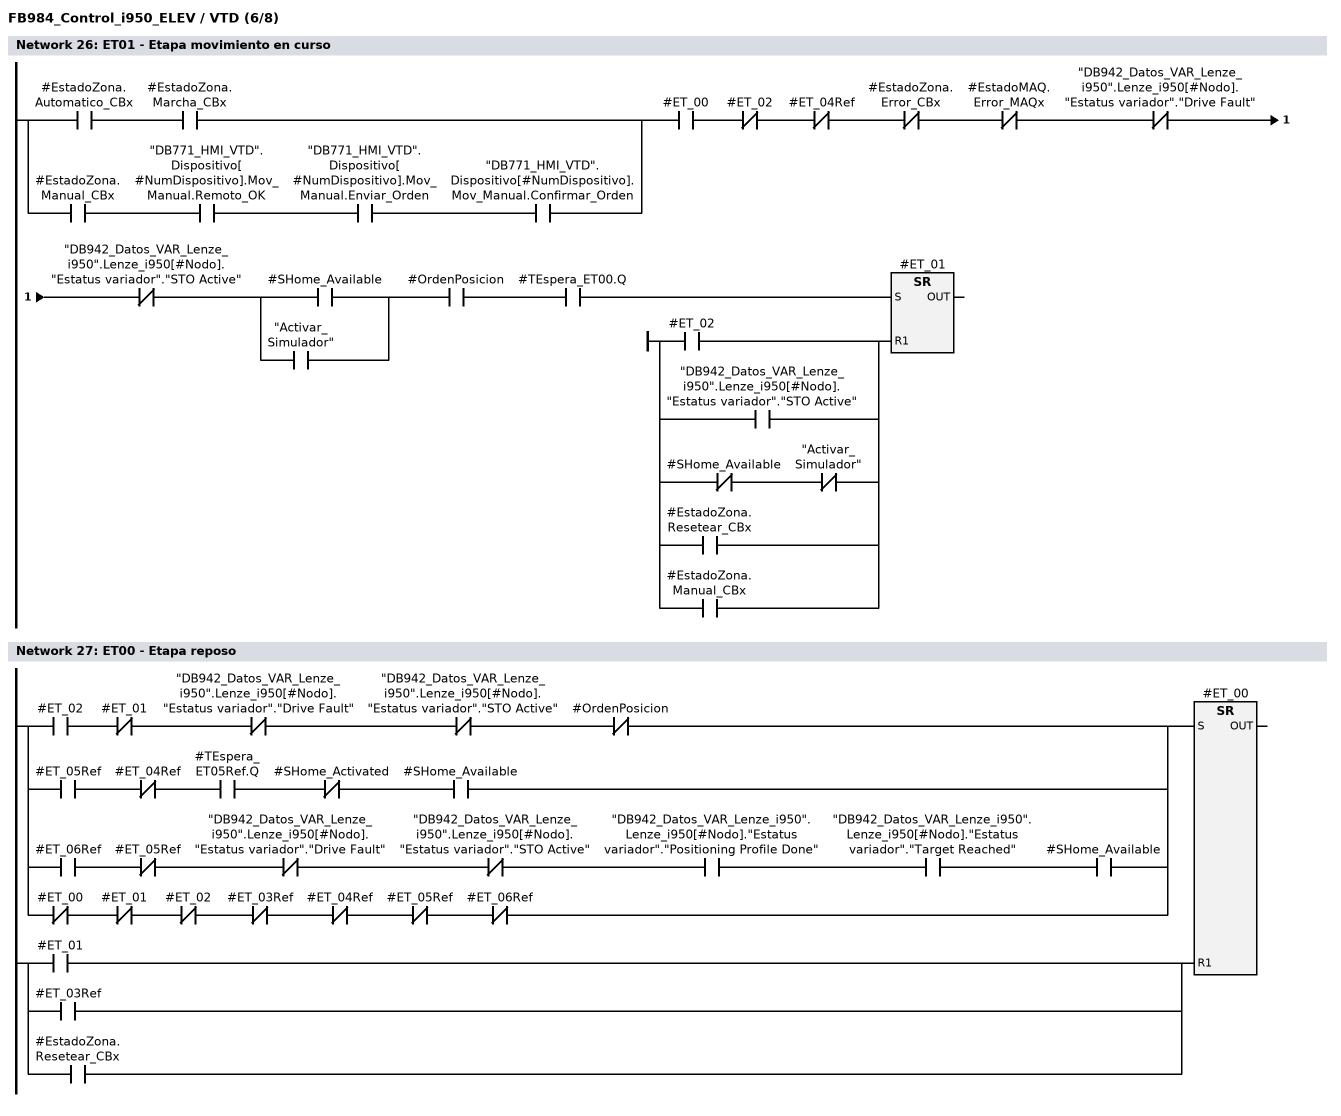
   RUNG wire#powerrail
      Contact( #EstadoZona.Automatico_CBx )
      Contact( #EstadoZona.Marcha_CBx )
      wire#w1
      Contact( #ET_00 )
      I_Contact( #ET_02 )
      I_Contact( #ET_04Ref )
      I_Contact( #EstadoZona.Error_CBx )
      I_Contact( #EstadoMAQ.Error_MAQx )
      I_Contact( "DB942_Datos_VAR_Lenze_i950".Lenze_i950[#Nodo]."Estatus variador"."Drive Fault" )
      I_Contact( "DB942_Datos_VAR_Lenze_i950".Lenze_i950[#Nodo]."Estatus variador"."STO Active" )
      wire#w2
      Contact( #SHome_Available )
      wire#w3
      Contact( #OrdenPosicion )
      Contact( #TEspera_ET00.Q )
      S_SR(operand := #ET_01, r1 := wire#w4)
   END_RUNG
   RUNG wire#powerrail
      Contact( #EstadoZona.Manual_CBx )
      Contact( "DB771_HMI_VTD".Dispositivo[#NumDispositivo].Mov_Manual.Remoto_OK )
      Contact( "DB771_HMI_VTD".Dispositivo[#NumDispositivo].Mov_Manual.Enviar_Orden )
      Contact( "DB771_HMI_VTD".Dispositivo[#NumDispositivo].Mov_Manual.Confirmar_Orden )
   END_RUNG wire#w1
   RUNG wire#w2
      Contact( "Activar_Simulador" )
   END_RUNG wire#w3
   RUNG wire#powerrail
      Contact( #ET_02 )
   END_RUNG wire#w4
   RUNG wire#powerrail
      Contact( "DB942_Datos_VAR_Lenze_i950".Lenze_i950[#Nodo]."Estatus variador"."STO Active" )
   END_RUNG wire#w4
   RUNG wire#powerrail
      I_Contact( #SHome_Available )
      I_Contact( "Activar_Simulador" )
   END_RUNG wire#w4
   RUNG wire#powerrail
      Contact( #EstadoZona.Resetear_CBx )
   END_RUNG wire#w4
   RUNG wire#powerrail
      Contact( #EstadoZona.Manual_CBx )
   END_RUNG wire#w4
   // the same network as SCL:
   IF ((#EstadoZona.Automatico_CBx AND #EstadoZona.Marcha_CBx) OR (#EstadoZona.Manual_CBx AND "DB771_HMI_VTD".Dispositivo[#NumDispositivo].Mov_Manual.Remoto_OK AND "DB771_HMI_VTD".Dispositivo[#NumDispositivo].Mov_Manual.Enviar_Orden AND "DB771_HMI_VTD".Dispositivo[#NumDispositivo].Mov_Manual.Confirmar_Orden)) AND #ET_00 AND NOT #ET_02 AND NOT #ET_04Ref AND NOT #EstadoZona.Error_CBx AND NOT #EstadoMAQ.Error_MAQx AND NOT "DB942_Datos_VAR_Lenze_i950".Lenze_i950[#Nodo]."Estatus variador"."Drive Fault" AND NOT "DB942_Datos_VAR_Lenze_i950".Lenze_i950[#Nodo]."Estatus variador"."STO Active" AND (#SHome_Available OR "Activar_Simulador") AND #OrdenPosicion AND #TEspera_ET00.Q THEN
       #ET_01 := TRUE;   // SR flip-flop
   END_IF;
   IF #ET_02 OR "DB942_Datos_VAR_Lenze_i950".Lenze_i950[#Nodo]."Estatus variador"."STO Active" OR (NOT #SHome_Available AND NOT "Activar_Simulador") OR #EstadoZona.Resetear_CBx OR #EstadoZona.Manual_CBx THEN
       #ET_01 := FALSE;
   END_IF;
END_REGION

REGION Network 27: ET00 - Etapa reposo
   RUNG wire#powerrail
      Contact( #ET_02 )
      I_Contact( #ET_01 )
      I_Contact( "DB942_Datos_VAR_Lenze_i950".Lenze_i950[#Nodo]."Estatus variador"."Drive Fault" )
      I_Contact( "DB942_Datos_VAR_Lenze_i950".Lenze_i950[#Nodo]."Estatus variador"."STO Active" )
      I_Contact( #OrdenPosicion )
      wire#w1
      S_SR(operand := #ET_00, r1 := wire#w2)
   END_RUNG
   RUNG wire#powerrail
      Contact( #ET_05Ref )
      I_Contact( #ET_04Ref )
      Contact( #TEspera_ET05Ref.Q )
      I_Contact( #SHome_Activated )
      Contact( #SHome_Available )
   END_RUNG wire#w1
   RUNG wire#powerrail
      Contact( #ET_06Ref )
      I_Contact( #ET_05Ref )
      I_Contact( "DB942_Datos_VAR_Lenze_i950".Lenze_i950[#Nodo]."Estatus variador"."Drive Fault" )
      I_Contact( "DB942_Datos_VAR_Lenze_i950".Lenze_i950[#Nodo]."Estatus variador"."STO Active" )
      Contact( "DB942_Datos_VAR_Lenze_i950".Lenze_i950[#Nodo]."Estatus variador"."Positioning Profile Done" )
      Contact( "DB942_Datos_VAR_Lenze_i950".Lenze_i950[#Nodo]."Estatus variador"."Target Reached" )
      Contact( #SHome_Available )
   END_RUNG wire#w1
   RUNG wire#powerrail
      I_Contact( #ET_00 )
      I_Contact( #ET_01 )
      I_Contact( #ET_02 )
      I_Contact( #ET_03Ref )
      I_Contact( #ET_04Ref )
      I_Contact( #ET_05Ref )
      I_Contact( #ET_06Ref )
   END_RUNG wire#w1
   RUNG wire#powerrail
      Contact( #ET_01 )
   END_RUNG wire#w2
   RUNG wire#powerrail
      Contact( #ET_03Ref )
   END_RUNG wire#w2
   RUNG wire#powerrail
      Contact( #EstadoZona.Resetear_CBx )
   END_RUNG wire#w2
   // the same network as SCL:
   IF (#ET_02 AND NOT #ET_01 AND NOT "DB942_Datos_VAR_Lenze_i950".Lenze_i950[#Nodo]."Estatus variador"."Drive Fault" AND NOT "DB942_Datos_VAR_Lenze_i950".Lenze_i950[#Nodo]."Estatus variador"."STO Active" AND NOT #OrdenPosicion) OR (#ET_05Ref AND NOT #ET_04Ref AND #TEspera_ET05Ref.Q AND NOT #SHome_Activated AND #SHome_Available) OR (#ET_06Ref AND NOT #ET_05Ref AND NOT "DB942_Datos_VAR_Lenze_i950".Lenze_i950[#Nodo]."Estatus variador"."Drive Fault" AND NOT "DB942_Datos_VAR_Lenze_i950".Lenze_i950[#Nodo]."Estatus variador"."STO Active" AND "DB942_Datos_VAR_Lenze_i950".Lenze_i950[#Nodo]."Estatus variador"."Positioning Profile Done" AND "DB942_Datos_VAR_Lenze_i950".Lenze_i950[#Nodo]."Estatus variador"."Target Reached" AND #SHome_Available) OR (NOT #ET_00 AND NOT #ET_01 AND NOT #ET_02 AND NOT #ET_03Ref AND NOT #ET_04Ref AND NOT #ET_05Ref AND NOT #ET_06Ref) THEN
       #ET_00 := TRUE;   // SR flip-flop
   END_IF;
   IF #ET_01 OR #ET_03Ref OR #EstadoZona.Resetear_CBx THEN #ET_00 := FALSE; END_IF;
END_REGION

REGION Network 28: >>>>>>>>>>>>>>>>>>>>>>>>>>>>>>>>>>>>>>>>>>>>>>>>>>>>>>>>>>>>>>>>>>>>>>>>>>>>>
END_REGION

REGION Network 29: Enable Operation
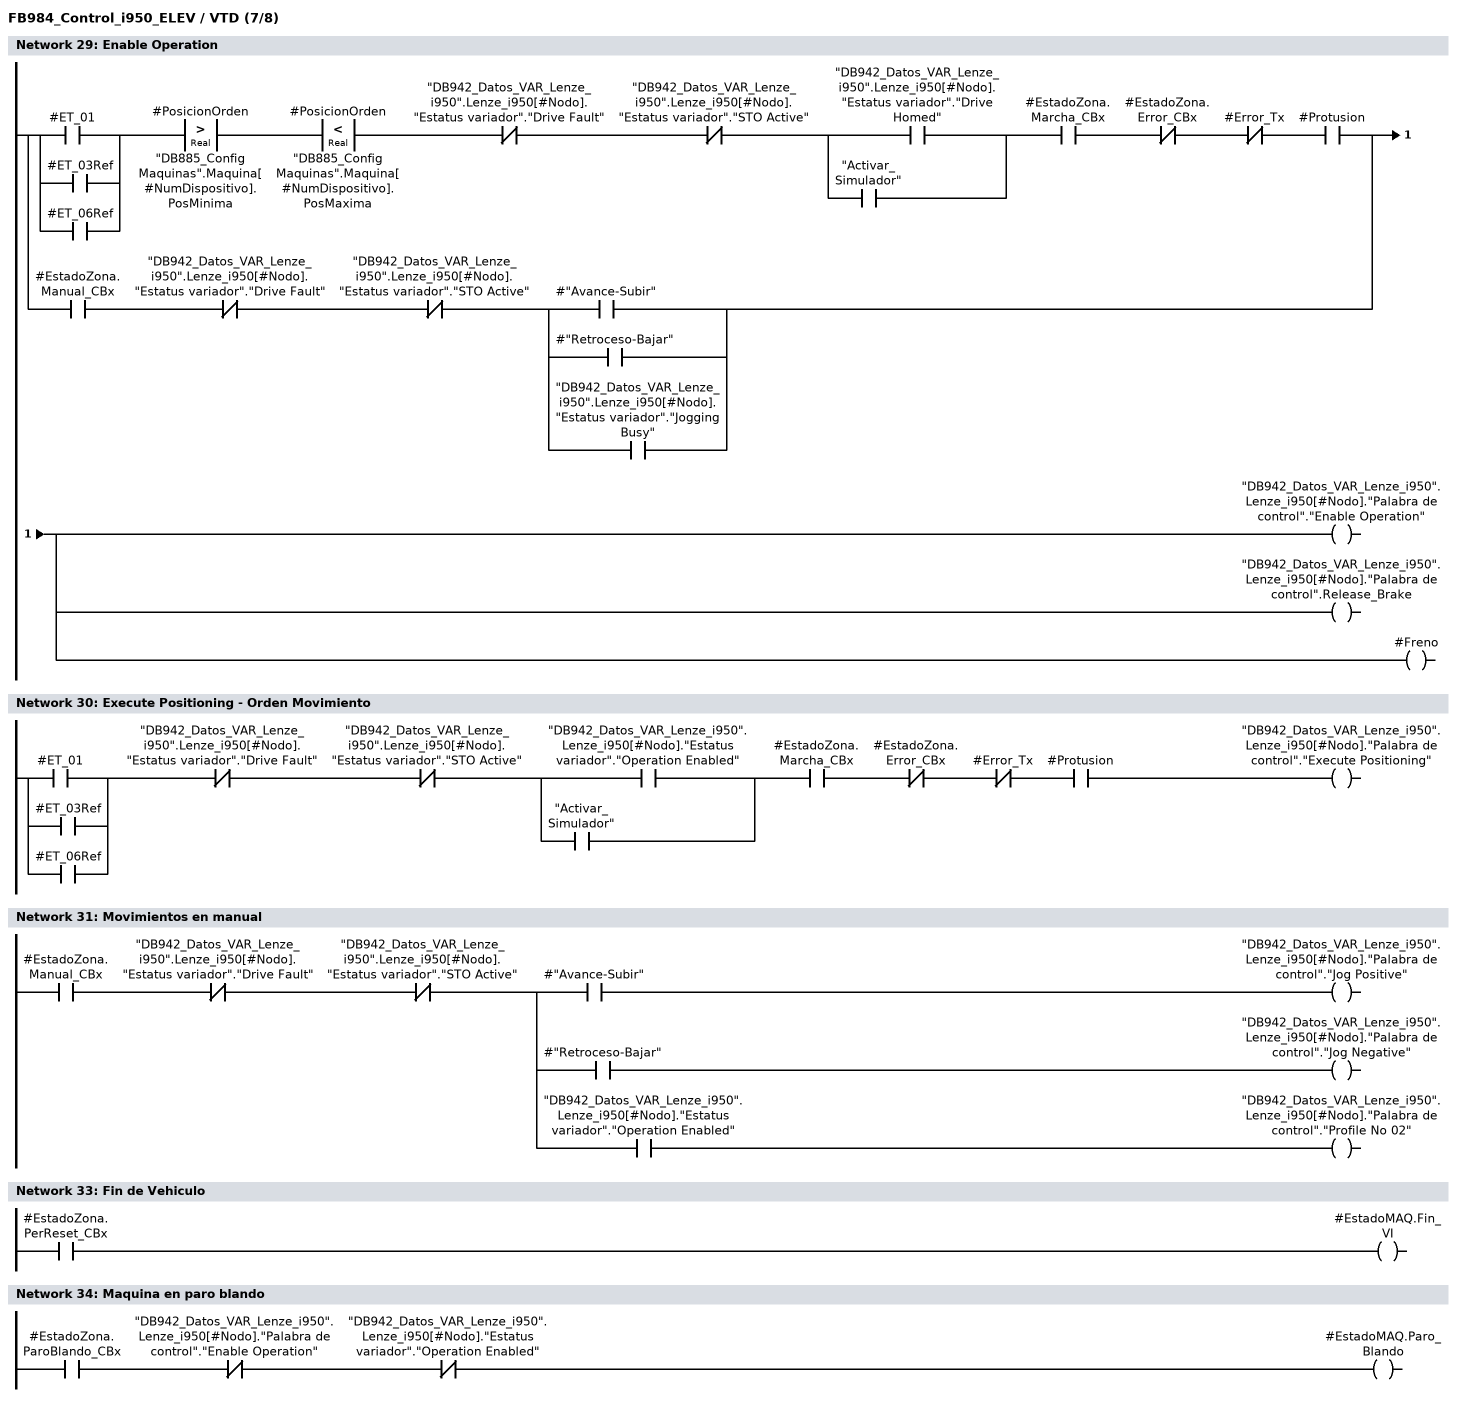
   RUNG wire#powerrail
      Contact( #ET_01 )
      wire#w1
      { S7_Templates := "SrcType := Real" } GT_Contact(in1 := #PosicionOrden, in2 := "DB885_ConfigMaquinas".Maquina[#NumDispositivo].PosMinima)
      { S7_Templates := "SrcType := Real" } LT_Contact(in1 := #PosicionOrden, in2 := "DB885_ConfigMaquinas".Maquina[#NumDispositivo].PosMaxima)
      I_Contact( "DB942_Datos_VAR_Lenze_i950".Lenze_i950[#Nodo]."Estatus variador"."Drive Fault" )
      I_Contact( "DB942_Datos_VAR_Lenze_i950".Lenze_i950[#Nodo]."Estatus variador"."STO Active" )
      wire#w2
      Contact( "DB942_Datos_VAR_Lenze_i950".Lenze_i950[#Nodo]."Estatus variador"."Drive Homed" )
      wire#w3
      Contact( #EstadoZona.Marcha_CBx )
      I_Contact( #EstadoZona.Error_CBx )
      I_Contact( #Error_Tx )
      Contact( #Protusion )
      wire#w4
      Coil( "DB942_Datos_VAR_Lenze_i950".Lenze_i950[#Nodo]."Palabra de control"."Enable Operation" )
   END_RUNG
   RUNG wire#powerrail
      Contact( #ET_03Ref )
   END_RUNG wire#w1
   RUNG wire#powerrail
      Contact( #ET_06Ref )
   END_RUNG wire#w1
   RUNG wire#w2
      Contact( "Activar_Simulador" )
   END_RUNG wire#w3
   RUNG wire#powerrail
      Contact( #EstadoZona.Manual_CBx )
      I_Contact( "DB942_Datos_VAR_Lenze_i950".Lenze_i950[#Nodo]."Estatus variador"."Drive Fault" )
      I_Contact( "DB942_Datos_VAR_Lenze_i950".Lenze_i950[#Nodo]."Estatus variador"."STO Active" )
      wire#w5
      Contact( #"Avance-Subir" )
   END_RUNG wire#w4
   RUNG wire#w5
      Contact( #"Retroceso-Bajar" )
   END_RUNG wire#w4
   RUNG wire#w5
      Contact( "DB942_Datos_VAR_Lenze_i950".Lenze_i950[#Nodo]."Estatus variador"."Jogging Busy" )
   END_RUNG wire#w4
   RUNG wire#w4
      Coil( "DB942_Datos_VAR_Lenze_i950".Lenze_i950[#Nodo]."Palabra de control".Release_Brake )
   END_RUNG
   RUNG wire#w4
      Coil( #Freno )
   END_RUNG
   // the same network as SCL:
   #_w1 := ((#ET_01 OR #ET_03Ref OR #ET_06Ref) AND (#PosicionOrden > "DB885_ConfigMaquinas".Maquina[#NumDispositivo].PosMinima) AND (#PosicionOrden < "DB885_ConfigMaquinas".Maquina[#NumDispositivo].PosMaxima) AND NOT "DB942_Datos_VAR_Lenze_i950".Lenze_i950[#Nodo]."Estatus variador"."Drive Fault" AND NOT "DB942_Datos_VAR_Lenze_i950".Lenze_i950[#Nodo]."Estatus variador"."STO Active" AND ("DB942_Datos_VAR_Lenze_i950".Lenze_i950[#Nodo]."Estatus variador"."Drive Homed" OR "Activar_Simulador") AND #EstadoZona.Marcha_CBx AND NOT #EstadoZona.Error_CBx AND NOT #Error_Tx AND #Protusion) OR (#EstadoZona.Manual_CBx AND NOT "DB942_Datos_VAR_Lenze_i950".Lenze_i950[#Nodo]."Estatus variador"."Drive Fault" AND NOT "DB942_Datos_VAR_Lenze_i950".Lenze_i950[#Nodo]."Estatus variador"."STO Active" AND (#"Avance-Subir" OR #"Retroceso-Bajar" OR "DB942_Datos_VAR_Lenze_i950".Lenze_i950[#Nodo]."Estatus variador"."Jogging Busy"));
   "DB942_Datos_VAR_Lenze_i950".Lenze_i950[#Nodo]."Palabra de control"."Enable Operation" := ((#ET_01 OR #ET_03Ref OR #ET_06Ref) AND (#PosicionOrden > "DB885_ConfigMaquinas".Maquina[#NumDispositivo].PosMinima) AND (#PosicionOrden < "DB885_ConfigMaquinas".Maquina[#NumDispositivo].PosMaxima) AND NOT "DB942_Datos_VAR_Lenze_i950".Lenze_i950[#Nodo]."Estatus variador"."Drive Fault" AND NOT "DB942_Datos_VAR_Lenze_i950".Lenze_i950[#Nodo]."Estatus variador"."STO Active" AND ("DB942_Datos_VAR_Lenze_i950".Lenze_i950[#Nodo]."Estatus variador"."Drive Homed" OR "Activar_Simulador") AND #EstadoZona.Marcha_CBx AND NOT #EstadoZona.Error_CBx AND NOT #Error_Tx AND #Protusion) OR (#EstadoZona.Manual_CBx AND NOT "DB942_Datos_VAR_Lenze_i950".Lenze_i950[#Nodo]."Estatus variador"."Drive Fault" AND NOT "DB942_Datos_VAR_Lenze_i950".Lenze_i950[#Nodo]."Estatus variador"."STO Active" AND (#"Avance-Subir" OR #"Retroceso-Bajar" OR "DB942_Datos_VAR_Lenze_i950".Lenze_i950[#Nodo]."Estatus variador"."Jogging Busy"));
   "DB942_Datos_VAR_Lenze_i950".Lenze_i950[#Nodo]."Palabra de control".Release_Brake := #_w1;
   #Freno := #_w1;
END_REGION

REGION Network 30: Execute Positioning - Orden Movimiento
   RUNG wire#powerrail
      Contact( #ET_01 )
      wire#w1
      I_Contact( "DB942_Datos_VAR_Lenze_i950".Lenze_i950[#Nodo]."Estatus variador"."Drive Fault" )
      I_Contact( "DB942_Datos_VAR_Lenze_i950".Lenze_i950[#Nodo]."Estatus variador"."STO Active" )
      wire#w2
      Contact( "DB942_Datos_VAR_Lenze_i950".Lenze_i950[#Nodo]."Estatus variador"."Operation Enabled" )
      wire#w3
      Contact( #EstadoZona.Marcha_CBx )
      I_Contact( #EstadoZona.Error_CBx )
      I_Contact( #Error_Tx )
      Contact( #Protusion )
      Coil( "DB942_Datos_VAR_Lenze_i950".Lenze_i950[#Nodo]."Palabra de control"."Execute Positioning" )
   END_RUNG
   RUNG wire#powerrail
      Contact( #ET_03Ref )
   END_RUNG wire#w1
   RUNG wire#powerrail
      Contact( #ET_06Ref )
   END_RUNG wire#w1
   RUNG wire#w2
      Contact( "Activar_Simulador" )
   END_RUNG wire#w3
   // the same network as SCL:
   "DB942_Datos_VAR_Lenze_i950".Lenze_i950[#Nodo]."Palabra de control"."Execute Positioning" := (#ET_01 OR #ET_03Ref OR #ET_06Ref) AND NOT "DB942_Datos_VAR_Lenze_i950".Lenze_i950[#Nodo]."Estatus variador"."Drive Fault" AND NOT "DB942_Datos_VAR_Lenze_i950".Lenze_i950[#Nodo]."Estatus variador"."STO Active" AND ("DB942_Datos_VAR_Lenze_i950".Lenze_i950[#Nodo]."Estatus variador"."Operation Enabled" OR "Activar_Simulador") AND #EstadoZona.Marcha_CBx AND NOT #EstadoZona.Error_CBx AND NOT #Error_Tx AND #Protusion;
END_REGION

REGION Network 31: Movimientos en manual
   RUNG wire#powerrail
      Contact( #EstadoZona.Manual_CBx )
      I_Contact( "DB942_Datos_VAR_Lenze_i950".Lenze_i950[#Nodo]."Estatus variador"."Drive Fault" )
      I_Contact( "DB942_Datos_VAR_Lenze_i950".Lenze_i950[#Nodo]."Estatus variador"."STO Active" )
      wire#w1
      Contact( #"Avance-Subir" )
      Coil( "DB942_Datos_VAR_Lenze_i950".Lenze_i950[#Nodo]."Palabra de control"."Jog Positive" )
   END_RUNG
   RUNG wire#w1
      Contact( #"Retroceso-Bajar" )
      Coil( "DB942_Datos_VAR_Lenze_i950".Lenze_i950[#Nodo]."Palabra de control"."Jog Negative" )
   END_RUNG
   RUNG wire#w1
      Contact( "DB942_Datos_VAR_Lenze_i950".Lenze_i950[#Nodo]."Estatus variador"."Operation Enabled" )
      Coil( "DB942_Datos_VAR_Lenze_i950".Lenze_i950[#Nodo]."Palabra de control"."Profile No 02" )
   END_RUNG
   // the same network as SCL:
   #_w1 := #EstadoZona.Manual_CBx AND NOT "DB942_Datos_VAR_Lenze_i950".Lenze_i950[#Nodo]."Estatus variador"."Drive Fault" AND NOT "DB942_Datos_VAR_Lenze_i950".Lenze_i950[#Nodo]."Estatus variador"."STO Active";
   "DB942_Datos_VAR_Lenze_i950".Lenze_i950[#Nodo]."Palabra de control"."Jog Positive" := #_w1 AND #"Avance-Subir";
   "DB942_Datos_VAR_Lenze_i950".Lenze_i950[#Nodo]."Palabra de control"."Jog Negative" := #_w1 AND #"Retroceso-Bajar";
   "DB942_Datos_VAR_Lenze_i950".Lenze_i950[#Nodo]."Palabra de control"."Profile No 02" := #_w1 AND "DB942_Datos_VAR_Lenze_i950".Lenze_i950[#Nodo]."Estatus variador"."Operation Enabled";
END_REGION

REGION Network 32 (SCL): Escritura variables al variador
   //Escribo las variables que nos interesan

   POKE_BOOL(area :=16#82,
             dbNumber :=0,
             byteOffset :=#Byte1,
             bitOffset :=0,
             value := "DB942_Datos_VAR_Lenze_i950".Lenze_i950[#Nodo]."Palabra de control"."Profile No 01");
   POKE_BOOL(area := 16#82,
             dbNumber := 0,
             byteOffset := #Byte0,
             bitOffset := 4,
             value :=  "DB942_Datos_VAR_Lenze_i950".Lenze_i950[#Nodo]."Palabra de control"."Activate Ext. Position");
   POKE_BOOL(area := 16#82,
             dbNumber := 0,
             byteOffset := #Byte0,
             bitOffset := 5,
             value := "DB942_Datos_VAR_Lenze_i950".Lenze_i950[#Nodo]."Palabra de control"."Activate Ext. Velocity");
   POKE_BOOL(area := 16#82,
             dbNumber := 0,
             byteOffset := #Byte0,
             bitOffset := 6,
             value := "DB942_Datos_VAR_Lenze_i950".Lenze_i950[#Nodo]."Palabra de control"."Activate Ext. Acc Dec Jerk");
   POKE_BOOL(area := 16#82,
             dbNumber := 0,
             byteOffset := #Byte1,
             bitOffset := 4,
             value := "DB942_Datos_VAR_Lenze_i950".Lenze_i950[#Nodo]."Palabra de control"."Execute Positioning");
   POKE_BOOL(area := 16#82,
             dbNumber := 0,
             byteOffset := #Byte2,
             bitOffset := 6,
             value := "DB942_Datos_VAR_Lenze_i950".Lenze_i950[#Nodo]."Palabra de control".Release_Brake);
   POKE_BOOL(area:= 16#82,
             dbNumber := 0,
             byteOffset := #Byte3,
             bitOffset := 3,
             value := "DB942_Datos_VAR_Lenze_i950".Lenze_i950[#Nodo]."Palabra de control"."Enable Operation");
   POKE_BOOL(area := 16#82,
             dbNumber := 0,
             byteOffset := #Byte3,
             bitOffset := 5,
             value := "DB942_Datos_VAR_Lenze_i950".Lenze_i950[#Nodo]."Palabra de control"."Jog Positive");
   POKE_BOOL(area := 16#82,
             dbNumber := 0,
             byteOffset := #Byte3,
             bitOffset := 6,
             value := "DB942_Datos_VAR_Lenze_i950".Lenze_i950[#Nodo]."Palabra de control"."Jog Negative");
   POKE_BOOL(area := 16#82,
             dbNumber := 0,
             byteOffset := #Byte3,
             bitOffset := 7,
             value := "DB942_Datos_VAR_Lenze_i950".Lenze_i950[#Nodo]."Palabra de control"."Fault Reset");


   POKE(area:=16#82,
        dbNumber:=0,
        byteOffset:=#Direccion_Velocity,
        value:= #ConsignaVelocidad);

   POKE(area := 16#82,
        dbNumber := 0,
        byteOffset := #Direccion_Position,
        value := "DB942_Datos_VAR_Lenze_i950".Lenze_i950[#Nodo].Target_Position);

   POKE(area := 16#82,
        dbNumber := 0,
        byteOffset := #Acele,
        value := "DB942_Datos_VAR_Lenze_i950".Lenze_i950[#Nodo].ACC);

   POKE(area := 16#82,
        dbNumber := 0,
        byteOffset := #Dece,
        value := "DB942_Datos_VAR_Lenze_i950".Lenze_i950[#Nodo].DCC);


   POKE(area := 16#82,
        dbNumber := 0,
        byteOffset := #Jerk,
        value := (#"VelocidadAuto(m/s)" * 300));

   POKE(area := 16#82,
        dbNumber := 0,
        byteOffset := #Torque,
        value := 0.0);
END_REGION

REGION Network 33: Fin de Vehiculo
   RUNG wire#powerrail
      Contact( #EstadoZona.PerReset_CBx )
      Coil( #EstadoMAQ.Fin_VI )
   END_RUNG
   // the same network as SCL:
   #EstadoMAQ.Fin_VI := #EstadoZona.PerReset_CBx;
END_REGION

REGION Network 34: Maquina en paro blando
   RUNG wire#powerrail
      Contact( #EstadoZona.ParoBlando_CBx )
      I_Contact( "DB942_Datos_VAR_Lenze_i950".Lenze_i950[#Nodo]."Palabra de control"."Enable Operation" )
      I_Contact( "DB942_Datos_VAR_Lenze_i950".Lenze_i950[#Nodo]."Estatus variador"."Operation Enabled" )
      Coil( #EstadoMAQ.Paro_Blando )
   END_RUNG
   // the same network as SCL:
   #EstadoMAQ.Paro_Blando := #EstadoZona.ParoBlando_CBx AND NOT "DB942_Datos_VAR_Lenze_i950".Lenze_i950[#Nodo]."Palabra de control"."Enable Operation" AND NOT "DB942_Datos_VAR_Lenze_i950".Lenze_i950[#Nodo]."Estatus variador"."Operation Enabled";
END_REGION

REGION Network 35: ERRORES
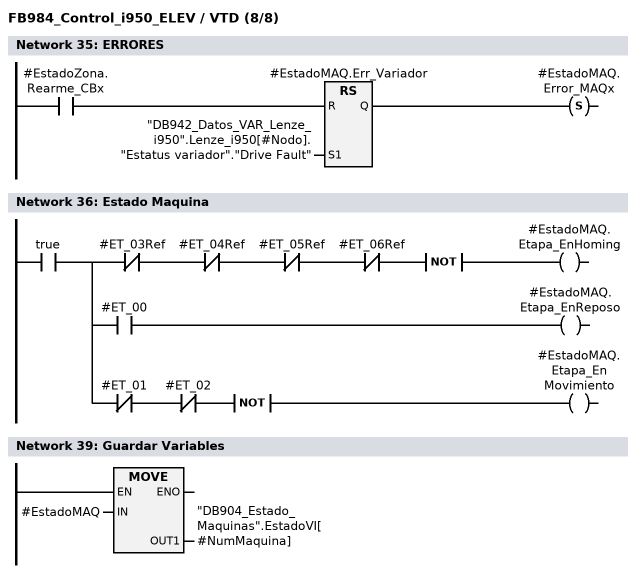
   RUNG wire#powerrail
      Contact( #EstadoZona.Rearme_CBx )
      S_RS(operand := #EstadoMAQ.Err_Variador, s1 := "DB942_Datos_VAR_Lenze_i950".Lenze_i950[#Nodo]."Estatus variador"."Drive Fault")
      S_Coil( #EstadoMAQ.Error_MAQx )
   END_RUNG
   // the same network as SCL:
   IF #EstadoZona.Rearme_CBx THEN
       #EstadoMAQ.Err_Variador := FALSE;   // RS flip-flop
   END_IF;
   IF "DB942_Datos_VAR_Lenze_i950".Lenze_i950[#Nodo]."Estatus variador"."Drive Fault" THEN
       #EstadoMAQ.Err_Variador := TRUE;
   END_IF;
   IF #EstadoMAQ.Err_Variador THEN #EstadoMAQ.Error_MAQx := TRUE; END_IF;
END_REGION

REGION Network 36: Estado Maquina
   RUNG wire#powerrail
      Contact( true )
      wire#w1
      I_Contact( #ET_03Ref )
      I_Contact( #ET_04Ref )
      I_Contact( #ET_05Ref )
      I_Contact( #ET_06Ref )
      Not()
      Coil( #EstadoMAQ.Etapa_EnHoming )
   END_RUNG
   RUNG wire#w1
      Contact( #ET_00 )
      Coil( #EstadoMAQ.Etapa_EnReposo )
   END_RUNG
   RUNG wire#w1
      I_Contact( #ET_01 )
      I_Contact( #ET_02 )
      Not()
      Coil( #EstadoMAQ.Etapa_EnMovimiento )
   END_RUNG
   // the same network as SCL:
   #EstadoMAQ.Etapa_EnHoming := NOT (true AND NOT #ET_03Ref AND NOT #ET_04Ref AND NOT #ET_05Ref AND NOT #ET_06Ref);
   #EstadoMAQ.Etapa_EnReposo := true AND #ET_00;
   #EstadoMAQ.Etapa_EnMovimiento := NOT (true AND NOT #ET_01 AND NOT #ET_02);
END_REGION

REGION Network 37 (SCL): VISUALIZACION
   "DB771_HMI_VTD".Dispositivo[#NumDispositivo].Estado_Variador."Estatus variador" := "DB942_Datos_VAR_Lenze_i950".Lenze_i950[#Nodo]."Estatus variador";
   "DB771_HMI_VTD".Dispositivo[#NumDispositivo].Estado_Variador."Palabra de control" := "DB942_Datos_VAR_Lenze_i950".Lenze_i950[#Nodo]."Palabra de control";
   "DB771_HMI_VTD".Dispositivo[#NumDispositivo].Estado_Variador."Código de error" := "DB942_Datos_VAR_Lenze_i950".Lenze_i950[#Nodo]."Código de error";
   "DB771_HMI_VTD".Dispositivo[#NumDispositivo].Position_Actual := DWORD_TO_DINT("DB942_Datos_VAR_Lenze_i950".Lenze_i950[#Nodo].Actual_Position);
   "DB771_HMI_VTD".Dispositivo[#NumDispositivo].Position_Destino := DWORD_TO_DINT("DB942_Datos_VAR_Lenze_i950".Lenze_i950[#Nodo].Target_Position);
   "DB771_HMI_VTD".Dispositivo[#NumDispositivo].EstadoVTD.Manual_CBx:=#EstadoMAQ.Manual;
   "DB771_HMI_VTD".Dispositivo[#NumDispositivo].EstadoVTD.Automatico_CBx := NOT #EstadoMAQ.Manual;
   "DB771_HMI_VTD".Dispositivo[#NumDispositivo].EstadoVTD.Marcha_CBx := #EstadoZona.Marcha_CBx;
END_REGION

REGION Network 38: >>>>>>>>>>>>>>>>>>>>>>>>>>>>>>>>>>>>>>>>>>>>>>>>>>>>>>>>>>>>>>>>>>>>>>>
END_REGION

REGION Network 39: Guardar Variables
   RUNG wire#powerrail
      Move(in := #EstadoMAQ, out1 => "DB904_Estado_Maquinas".EstadoVI[#NumMaquina])
   END_RUNG
   // the same network as SCL:
   "DB904_Estado_Maquinas".EstadoVI[#NumMaquina] := #EstadoMAQ;
END_REGION
END_FUNCTION_BLOCK
